(* PLC project boxtri, Dassault Systèmes ControlBuild 2024x *)
(* stored: creationDateTime 2023-10-03T11:14:00-01:00 *)

FUNCTION_BLOCK tri_chain.boxtri
  VAR
    status_act_prod : DINT := 0;
    m11 : REAL := 1.0;
    m12 : REAL := 0.0;
    m13 : REAL := 0.0;
    m14 : REAL := 0.0;
    m21 : REAL := 0.0;
    m22 : REAL := 1.0;
    m23 : REAL := 0.0;
    m24 : REAL := 0.0;
    m31 : REAL := 0.0;
    m32 : REAL := 0.0;
    m33 : REAL := 1.0;
    m34 : REAL := 0.0;
    m41 : REAL := 0.0;
    m42 : REAL := 0.0;
    m43 : REAL := 0.0;
    m44 : REAL := 1.0;
    px : REAL := 0.0;
    py : REAL := 0.0;
    pz : REAL := 0.0;
    dx : REAL := 0.0;
    dy : REAL := 0.0;
    dz : REAL := 0.0;
    sxInter : REAL := 0.0;
    syInter : REAL := 0.0;
    interacNb : REAL := 0.0;
  END_VAR


ACTION Prelude:
interacNb = 0.0;
sxInter = 0.0;
syInter = 0.0;


px = getPositionX(myself);
py = getPositionY(myself);
pz = getPositionZ(myself);

dx = getDX(myself);
dy = getDY(myself);
dz = getDZ(myself);
END_ACTION

ACTION Postlude:
if (interacNb > 0.0) syInter = syInter / interacNb;
else syInter = 0.0;

if (syInter != 0.0) sxInter = syInter * (-0.25);
px = px + sxInter;
py = py - syInter;




moveTo(myself, px, py, pz);
END_ACTION

ACTION tri_chain.shuttle:
syInter = syInter + otherVar(sProdY);
sxInter = otherVar(sProdX);
interacNb = interacNb + 1.0;
END_ACTION

ACTION tri_chain.passing_sensor:
otherVar(detection)=1;
END_ACTION

ACTION tri_chain.passing_sensor2:
otherVar(detection)=1;
END_ACTION

ACTION tri_chain.creation:
otherVar(presenceProduct)=1;
END_ACTION

ACTION tri_chain.trash:
prodKill(myself);
END_ACTION

ACTION tri_chain.conveyor1:
syInter = syInter + otherVar(sProduct);
interacNb = interacNb + 1.0;

otherVar(interaction) = 1;
END_ACTION
END_FUNCTION_BLOCK
